(* Schneider Machine Expert - Basic project tank_level_control_TM221CE16T, file version 3.0.0.0 *)
(* ProjectInformations: Name=Tank Level Control TM221CE16T with TM3AI4 *)

HARDWARE
  Cpu 0: TM221CE16T
  Extension 0: TM3AI4
  EthernetConfiguration: NetworkName=M221, IpAllocationMode=ByDhcp, IpAddress=192.168.1.10, SubnetMask=255.255.255.0
  SerialLineConfiguration: Baud=Baud19200, Parity=ParityEven, DataBits=DataBits8, StopBits=StopBits1, PhysicalMedium=PhysicalMediumRs485, TransmissionMode=TransmissionModeModbusRtu, SlaveId=1, Addressing=SlaveAddressing
  MastTask: UsePeriodScanMode=false, PeriodScan=100
  FastTask: Period=255
  CpuBehavior: StartingMode=StartAsPreviousState, AutoSaveRamOnEeprom=true, WatchdogPeriod=250

SYMBOLS  (address, symbol, comment, settings)
  %M0       TANK_FULL  "Tank full flag from ultrasonic sensor"
  %M1       TANK_EMPTY  "Tank empty flag from ultrasonic sensor"
  %Q0.0     INLET_VLV  "Inlet valve solenoid"
  %Q0.1     OUTLET_VLV  "Outlet valve solenoid"
  %IW1.0    LEVEL_AIN  "Ultrasonic level transmitter 4-20mA"  [AIType=Current4_20mA, AIRange=Range0_10000, AIFilter=AIFilter4]

POU Tank Level Control
  (* SectionNumber=1 *)

// Rung 0: Tank Full Detection
// Ultrasonic sensor: low value means tank is full. Set flag when level reading below 1800.
  LD [%IW1.0<1800]        (* LEVEL_AIN *)
  ST %M0                  (* TANK_FULL *)
  // as ST:
  //   TANK_FULL := LEVEL_AIN<1800;
  (* the ladder stored for this rung does not match its IL; not drawn *)

// Rung 1: Tank Empty Detection
// Ultrasonic sensor: high value means tank is empty. Set flag when level reading above 4800.
  LD [%IW1.0>4800]        (* LEVEL_AIN *)
  ST %M1                  (* TANK_EMPTY *)
  // as ST:
  //   TANK_EMPTY := LEVEL_AIN>4800;
  (* the ladder stored for this rung does not match its IL; not drawn *)

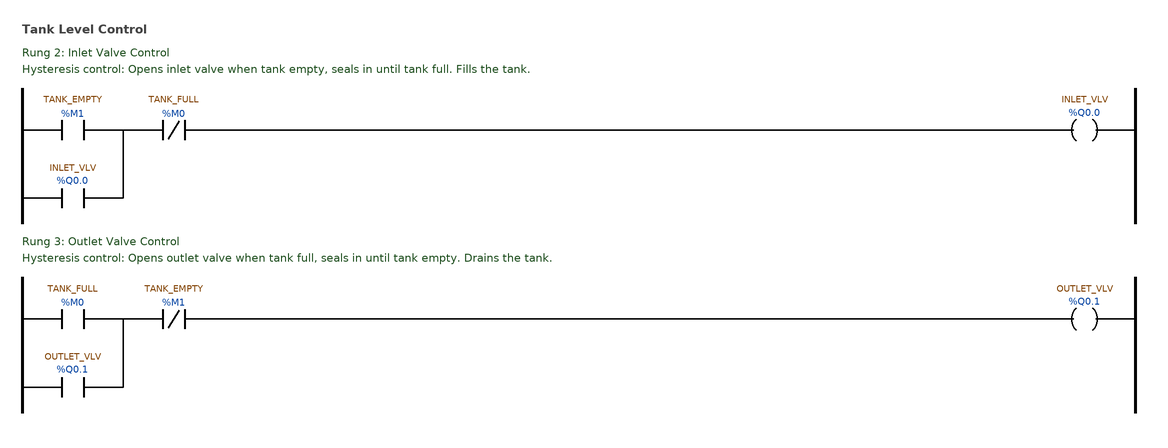

// Rung 2: Inlet Valve Control
// Hysteresis control: Opens inlet valve when tank empty, seals in until tank full. Fills the tank.
  LD %M1                  (* TANK_EMPTY *)
  OR %Q0.0                (* INLET_VLV *)
  ANDN %M0                (* TANK_FULL *)
  ST %Q0.0                (* INLET_VLV *)
  // as ST:
  //   INLET_VLV := (TANK_EMPTY OR INLET_VLV) AND NOT TANK_FULL;

// Rung 3: Outlet Valve Control
// Hysteresis control: Opens outlet valve when tank full, seals in until tank empty. Drains the tank.
  LD %M0                  (* TANK_FULL *)
  OR %Q0.1                (* OUTLET_VLV *)
  ANDN %M1                (* TANK_EMPTY *)
  ST %Q0.1                (* OUTLET_VLV *)
  // as ST:
  //   OUTLET_VLV := (TANK_FULL OR OUTLET_VLV) AND NOT TANK_EMPTY;
